{attribute 'GeneratedUsingTerminal: EL5151-0000-0017'}
{attribute addProperty BoxType "EL5151-0000-0017"}
{attribute addProperty Id "ENC_InputsAT %I*ENC_Inputs_561E041F18ENC_Inputs_1AT %I*ENC_Inputs_24B63C534ENC_OutputsAT %Q*ENC_Outputs_2E45048F8WcStateAT %I*WcState_9091E0EB2InfoDataAT %I*InfoData_94A18F5E2"}
{attribute addProperty CRC "1940515144"}
{attribute addProperty Size "34"}
TYPE EL5151_73A9E948 EXTENDS EtcSlaveTerminalBase_947E5A46 :
STRUCT
	{attribute addProperty Name "ENC_Inputs"}
	ENC_Inputs : ENC_Inputs_561E041F;
	{attribute addProperty Name "ENC_Inputs_1"}
	ENC_Inputs_1 : ENC_Inputs_24B63C53;
	{attribute addProperty Name "ENC_Outputs"}
	ENC_Outputs : ENC_Outputs_2E45048F;
	{attribute addProperty Name "WcState"}
	WcState : WcState_9091E0EB;
	{attribute addProperty Name "InfoData"}
	InfoData : InfoData_94A18F5E;
END_STRUCT
END_TYPE

(* stored: Version 1.2.0.0, ProductVersion 3.1.4024.9
   DUT EL5151_73A9E948: Id {9702795b-1e69-4f8a-bd77-19136c438114} *)
